// TIA Portal project "学习OB100和OB" (V16)

(* hardware
DEVICE "S7-1200 station_1"  S7-1200 Station
   slot 0: "Rack_0"  S7-1200 Rack  Rack  V1.0
   slot 1: "PLC_1"  CPU 1214C DC/DC/Rly  6ES7 214-1HG40-0XB0  V4.4
*)

// ===== PLC "PLC_1"  CPU 1214C DC/DC/Rly =====

VAR_GLOBAL   // PLC tag table "默认变量表"
   "Tag_1" AT %MW100 : Int;
   "Tag_2" AT %MW12 : Int;
   "Tag_3" AT %MW4 : Int;
   "Tag_4" AT %MW6 : Int;
   "Tag_5" AT %MW16 : Word;
END_VAR

ORGANIZATION_BLOCK "Main"   // OB1, LAD, ProgramCycle
TITLE = "Main Program Sweep (Cycle)"
{ S7_Optimized_Access := 'TRUE' }
VERSION : 0.1
   VAR_INPUT
      Initial_Call : Bool;   // Initial call of this OB
      Remanence : Bool;   // =True, if remanent data are available
   END_VAR
BEGIN
END_ORGANIZATION_BLOCK

ORGANIZATION_BLOCK "循环100ms"   // OB30, LAD, CyclicInterrupt
{ S7_Optimized_Access := 'TRUE' }
VERSION : 0.1
   VAR_INPUT
      Initial_Call : Bool;   // Initial call of this OB
      Event_Count : Int;   // Events discarded
   END_VAR
BEGIN

REGION Network 1
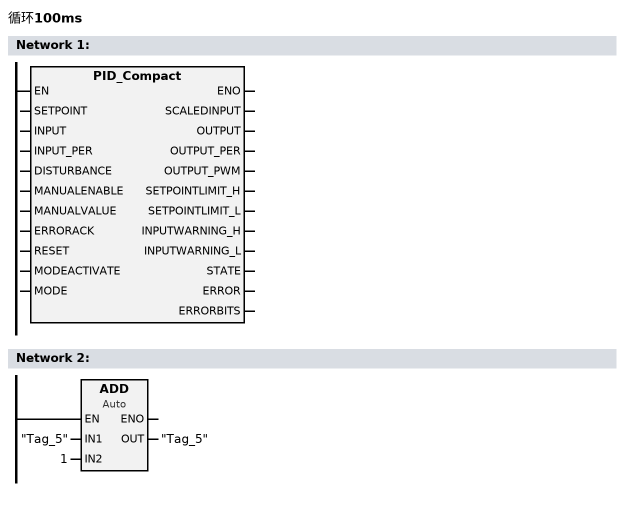
   // no SCL statement known for PID_Compact: written as a call
   PID_Compact();
END_REGION

REGION Network 2
   RUNG wire#powerrail
      Add(in1 := "Tag_5", in2 := 1, out => "Tag_5")
   END_RUNG
   // the same network as SCL:
   "Tag_5" := "Tag_5" + 1;
END_REGION
END_ORGANIZATION_BLOCK

ORGANIZATION_BLOCK "Startup"   // OB100, LAD, Startup
TITLE = "Complete Restart"
{ S7_Optimized_Access := 'TRUE' }
VERSION : 0.1
   VAR_INPUT
      LostRetentive : Bool;   // True if retentive data are lost
      LostRTC : Bool;   // True if date and time are lost
   END_VAR
BEGIN

REGION Network 1
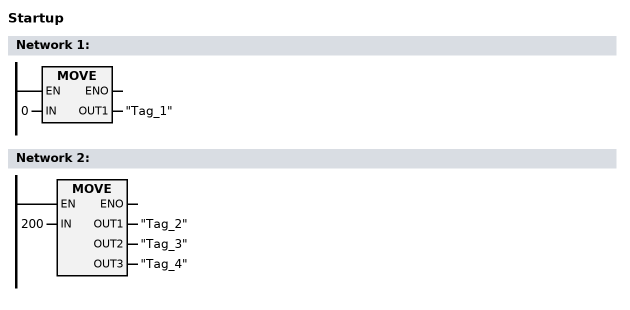
   RUNG wire#powerrail
      Move(in := 0, out1 => "Tag_1")
   END_RUNG
   // the same network as SCL:
   "Tag_1" := 0;
END_REGION

REGION Network 2
   RUNG wire#powerrail
      Move(in := 200, out1 => "Tag_2", out2 => "Tag_3", out3 => "Tag_4")
   END_RUNG
   // the same network as SCL:
   "Tag_2" := 200;
   "Tag_3" := 200;
   "Tag_4" := 200;
END_REGION
END_ORGANIZATION_BLOCK